// TIA Portal V17 export
// export: Created 2024-01-30T08:49:17.0389622Z, ExportSetting WithDefaults, DisplayName Totally Integrated Automation Portal, DisplayVersion V17 Update 6, DisplayName TIA Portal Openness, DisplayVersion V17 Update 6, DisplayName TIA Portal Version Control Interface, DisplayVersion V17, DisplayName STEP 7 Professional, DisplayVersion V17 Update 6, DisplayName STEP 7 Safety, DisplayVersion V17 Update 6, DisplayName WinCC Advanced, DisplayVersion V17 Update 6
TYPE "TRACKING_SYSTEM_TEMPOPC"
// stored: IsFailsafeCompliant false
   STRUCT
      MainDB : "OvenTemperature";
      Req_Start { S7_SetPoint := 'True'} : Bool;
      Archive_Done : Bool;
   END_STRUCT;
END_TYPE
